{attribute 'GeneratedUsingTerminal: EJ2522-0000-0022'}
{attribute addProperty BoxType "EJ2522-0000-0022"}
{attribute addProperty Id "ControlAT %Q*Control_A8DDCD822Set_counter_valueAT %Q*UDINT4"}
{attribute addProperty CRC "1751890396"}
{attribute addProperty Size "6"}
TYPE ENC_Control_Channel_686BB9DC EXTENDS OutputBase_10CEE7DE :
STRUCT
	{attribute addProperty Name "Control"}
	Control AT %Q* : Control_A8DDCD82;
	{attribute addProperty Name "Set_counter_value"}
	Set_counter_value AT %Q* : UDINT;
END_STRUCT
END_TYPE
